PROGRAM MAIN
VAR
END_VAR

END_PROGRAM

(* stored: Version 1.1.0.1
   POU MAIN: Id {5ea970d2-a3c2-417b-b85f-4fd77acaeb11} *)
